// TIA Portal V20 export
ORGANIZATION_BLOCK "Main"   // OB126, LAD, ProgramCycle
TITLE = "Main Program Sweep (Cycle)"
// stored: Namespace Conveyor4, SetENOAutomatically false
   VAR_INPUT
      Initial_Call : Bool;   // Initial call of this OB
      Remanence : Bool;   // =True, if remanent data are available
   END_VAR
BEGIN

REGION Network 1
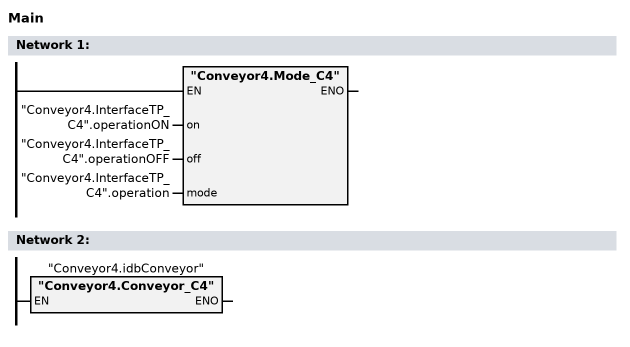
   RUNG wire#powerrail
      "Conveyor4.Mode_C4"(on := "Conveyor4.InterfaceTP_C4".operationON, off := "Conveyor4.InterfaceTP_C4".operationOFF, mode := "Conveyor4.InterfaceTP_C4".operation)
   END_RUNG
   // the same network as SCL:
   "Conveyor4.Mode_C4"(on := "Conveyor4.InterfaceTP_C4".operationON,
                       off := "Conveyor4.InterfaceTP_C4".operationOFF,
                       mode := "Conveyor4.InterfaceTP_C4".operation);
END_REGION

REGION Network 2
   RUNG wire#powerrail
      "Conveyor4.idbConveyor"()
   END_RUNG
   // the same network as SCL:
   "Conveyor4.idbConveyor"();   // "Conveyor4.Conveyor_C4"
END_REGION
END_ORGANIZATION_BLOCK
